PROGRAM MAIN
VAR
END_VAR

END_PROGRAM

(* stored: Version 1.1.0.1
   POU MAIN: Id {df34335a-3519-4b7e-97b2-e9631f15eddb} *)
